(*

short summary
=============
dispather for lollipops

legal notes
===========
SPDX-FileCopyrightText: © 2024 ekvip automation GmbH <info@ekvip.de>
SPDX-License-Identifier: Apache-2.0
For details check: Apache-2.0_

.. _Apache-2.0: https://www.apache.org/licenses/LICENSE-2.0

*)

{attribute 'enable_dynamic_creation'}
FUNCTION_BLOCK FINAL LollipopsDispatcher EXTENDS AbstractCandyDispatcher

(*

short summary
=============
this method dispatches lollipops
to a candy consumer 

legal notes
===========
SPDX-FileCopyrightText: © 2024 ekvip automation GmbH <info@ekvip.de>
SPDX-License-Identifier: Apache-2.0
For details check: Apache-2.0_

.. _Apache-2.0: https://www.apache.org/licenses/LICENSE-2.0

*)

METHOD eat
VAR_INPUT
	(* consumer who eats the candy *)
	consumer	:REFERENCE TO AbstractCandyConsumer;
	(* candy amount in gram *)
	amount		:CandyAmountInGram;
END_VAR
RETURN(THIS^.eatCandiesIsImpossible(consumer, amount));
consumer.eatLollipops(amount);
END_METHOD

END_FUNCTION_BLOCK

(* stored: Version 1.1.0.1
   POU LollipopsDispatcher: Id {e08364af-75ff-472d-8c01-3770a103148f}, SpecialFunc None
   Method eat: Id {ee26dfae-1947-4885-81a9-d66c5be34afe} *)
